INTERFACE I_MachiningExecutor

METHOD Abort
VAR_INPUT
END_VAR
END_METHOD

PROPERTY Busy : BOOL
GET
END_GET
END_PROPERTY

PROPERTY Done : BOOL
GET
END_GET
END_PROPERTY

PROPERTY Error : BOOL
GET
END_GET
END_PROPERTY

PROPERTY ErrorID : UDINT
GET
END_GET
END_PROPERTY

METHOD Execute : BOOL
VAR_INPUT
END_VAR
END_METHOD

END_INTERFACE

(* stored: Version 1.1.0.1, ProductVersion 3.1.4024.15
   Itf I_MachiningExecutor: Id {5c743b52-4b22-4c04-8775-ad733b78e5a4}
   Method Abort: Id {21640305-90fb-40a8-9fa4-675e9a875812}
   Property Busy: Id {acba1e1c-8eeb-46cc-89c2-4e9c098c53e2}
   Get Get: Id {0454df02-f219-4838-93d7-84edb612c046}
   Property Done: Id {6a19729a-dd40-4291-8863-4445469a4472}
   Get Get: Id {cbcf412b-07ee-4636-897f-76aa76d67693}
   Property Error: Id {663a4edc-2c42-4f65-a14b-4a6081319b3a}
   Get Get: Id {7a925b2c-c7e6-4959-a708-2b27f3822c0e}
   Property ErrorID: Id {0345e46d-dd68-4f63-9243-5314ca13c2e5}
   Get Get: Id {54beebcb-f22c-49ca-bd3d-4693796d87e4}
   Method Execute: Id {c3dc2c55-7d23-4aed-9215-6c671f3e34d6} *)
